PROGRAM PRG_INIT
VAR
	init: INT;
	initEdge : R_TRIG;
END_VAR

//ob pritisku na Init tipko gre v izhodisce
initEdge(CLK:=IO.bInit);


CASE init OF
	0:
		IF initEdge.Q AND (main.iKorak <> 50) THEN
		MAIN.iKorak := -1;
		
		END_IF;
		init := 10;
	10:
		
		IF (main.iKorak = 50) AND initEdge.Q THEN	
			MAIN.iKorakRelativnegaPomika := -1;
		END_IF
	
		IF main.iKorak = 100 THEN
			init := 0;
		END_IF
	
END_CASE

END_PROGRAM

(* stored: Version 1.1.0.1, ProductVersion 3.1.4024.9
   POU PRG_INIT: Id {5483ec78-59fd-4af6-a1b4-63ebbd26ad06}, SpecialFunc None *)
